FUNCTION FC_MEMCPY_FLIP_WORD : BOOL
VAR_IN_OUT
	Source : ARRAY[*] OF BYTE;
END_VAR
VAR_INPUT
	Dest : POINTER TO BYTE;
END_VAR
VAR
	ArrLen : UDINT;
	NewArray : POINTER TO BYTE;
	i : DINT;
	Overflow : DINT;
END_VAR

ArrLen := DINT_TO_UDINT((UPPER_BOUND(Source,1) - LOWER_BOUND(Source,1)) + 1);

NewArray := __NEW(BYTE, ArrLen);
Overflow := UDINT_TO_DINT(ArrLen MOD 4);

FOR i := LOWER_BOUND(Source,1) TO UPPER_BOUND(Source,1) BY 4 DO
	IF i < (UPPER_BOUND(Source,1) - Overflow) THEN
		NewArray[i] := Source[i + 3];
		NewArray[i + 1] := Source[i + 2];
		NewArray[i + 2] := Source[i + 1];
		NewArray[i + 3] := Source[i];
	ELSE
		NewArray[i] := Source[i];
	END_IF;
END_FOR;

MEMCPY(Dest, NewArray, ArrLen);

__DELETE(NewArray);

END_FUNCTION

(* stored: Version 1.1.0.1, ProductVersion 3.1.4024.12
   POU FC_MEMCPY_FLIP_WORD: Id {5919394a-bf09-4025-a77b-5dae90416827}, SpecialFunc None *)
